// TIA Portal project "Tesis_Aeroponicos_V1" (V15.1)

(* hardware
DEVICE "S7300/ET200M station_1"  S7-300 station
   slot 0: "Rail_0"  Rail  6ES7 390-1***0-0AA0
   slot 2: "PLC_1"  CPU 313C  6ES7 313-5BF03-0AB0  V2.6
      slot 0: "MPI interface_1"  X1
      slot 2: "DI 24/DO 16_1"  DI24/DO16
      slot 3: "AI 5/AO 2_1"  AI5/AO2
      slot 4: "Count_1"  Counter
   slot 4: "CP 343-1 Advanced-IT_1"  CP 343-1 ADVANCED-IT  6GK7 343-1GX30-0XE0  V1.2
*)

// ===== PLC "PLC_1"  CPU 313C =====

VAR_GLOBAL   // PLC tag table "Default tag table"
   "E/S LoRa" AT %IW752 : Int;
   "E/S Valvula" AT %QW752 : Int;
   "D_valvula" AT %Q124.0 : Bool;
   "IO_1" AT %I124.0 : Bool;
   "Tag_1" AT %MW1 : Int;
   "Salida" AT %MD4 : Real;
   "Flag2" AT %M0.0 : Bool;
   "Entero" AT %MW8 : Int;
   "Tag_2" AT %M0.1 : Bool;
   "Test" AT %Q124.1 : Bool;
   "Control_temp" AT %Q125.7 : Bool;
   "Tag_3" AT %MD12 : Real;
   "Riego_45" AT %Q125.6 : Bool;
   "Riego_30" AT %Q125.5 : Bool;
   "Riego_15" AT %Q125.4 : Bool;
   "Tag_4" AT %T0 : Timer;
   "Tag_5" AT %T1 : Timer;
   "Tag_6" AT %M0.2 : Bool;
   "Tag_7" AT %M0.3 : Bool;
   "Tag_8" AT %M0.4 : Bool;
   "Tag_9" AT %M0.5 : Bool;
   "Tag_10" AT %T2 : Timer;
   "Tag_11" AT %T3 : Timer;
   "Tag_12" AT %MW6 : Word;
   "Tag_13" AT %M0.6 : Bool;
   "Tag_14" AT %M0.7 : Bool;
END_VAR

// folder: SystemBlocksFolder/ReportSystemErrorFolder

DATA_BLOCK "RSE_DIAGNOSTIC_STATUS_DB"   // DB127
TITLE = Bloque de diagnóstico Notificar errores del sistema
{ S7_Optimized_Access := 'FALSE' }
AUTHOR : SIMATIC
FAMILY : RSEDIAG
NAME : RSE7
VERSION : 1.0
// Este DB forma parte de Notificar errores de sistema y es actualizado por el FB de Notificar errores de sistema.
//  Es una interfaz para asistir el diagnóstico de sistema a través del CPU Webserver.
   VAR
      Directory : Struct
         D_Version : Word := WORD#16#0100;   // Versión que soporta 'Notificar errores de sistema' (SFM)
         D_pGlobalState : Word := WORD#16#0010;   // Offset de byte hasta el principio de la parte "GlobalState"
         D_pQuery : Word := WORD#16#0014;   // Offset de byte hasta el principio de la parte "Query"
         D_pComponent : Word := WORD#16#0020;   // Offset de byte hasta el principio de la parte "Component"
         D_pError : Word := WORD#16#0024;   // Offset de byte hasta el principio de la parte "Error"
         D_pState : Word := WORD#16#0028;   // Offset de byte hasta el principio de la parte "State"
         D_pAlarm : Word := WORD#16#005A;   // Offset de byte hasta el principio de la parte "Alarm"
         D_pSubComponent : Word := WORD#16#0082;   // Offset de byte hasta el principio de la parte "Subcomponent"
      END_STRUCT;
      GlobalState : Struct
         G_EventCount : Word := WORD#16#0000;   // ID del último evento (contador)
         G_StartReporting : Bool := FALSE;   // Evaluando el arranque
      END_STRUCT;
      Query : Struct
         Q_ClientID_User : DWord := DWORD#16#0000_0000;   // ID del cliente
         Q_ClientID_Intern : DWord := DWORD#16#0000_0000;   // ID del cliente (interno)
         Q_WithSubComponent : Bool := FALSE;   // Con/sin estado de los subcomponentes (más lento)
         Q_SubComponentAlarm : Bool := FALSE;   // AS-iMaster gibt AS-iSlave Alarme zurück
         Q_Reserved2 : Bool := FALSE;   // Reservado
         Q_Reserved3 : Bool := FALSE;   // Reservado
         Q_Reserved4 : Bool := FALSE;   // Reservado
         Q_Reserved5 : Bool := FALSE;   // Reservado
         Q_Reserved6 : Bool := FALSE;   // Reservado
         Q_Reserved7 : Bool := FALSE;   // Reservado
         Q_Start : Bool := FALSE;   // Iniciar consulta
         Q_Error : Byte := BYTE#16#00;   // Error interno en la consulta
         Q_Reserved8 : Byte := BYTE#16#00;   // Reservado
      END_STRUCT;
      Component : Struct
         C_AddressMode : Byte := BYTE#16#00;   // Modo de direccionamiento del módulo
         C_Reserved1 : Byte := BYTE#16#00;   // Reservado
         C_ComponentID : Word := WORD#16#0000;   // ID de hardware del componente (interno)
      END_STRUCT;
      Error : Struct
         E_ErrorNo : Word := WORD#16#0000;   // Índice del error solicitado/efectivo
         E_LastError : Bool := FALSE;   // TRUE, si E_ErrorNo contiene el índice del último error, de lo contrario FALSE
      END_STRUCT;
      State : Struct
         S_Hierarchy : Byte := BYTE#16#00;   // Reservado
         S_Periphery : Byte := BYTE#16#00;   // Reservado
         S_SupFault : Bool := FALSE;   // No se puede acceder al componente
         S_NotAvailable : Bool := FALSE;   // El componente no existe
         S_Faulty : Bool := FALSE;   // El componente falla; la parte "Alarm" no está vacía
         S_MoreErrors : Bool := FALSE;   // Hay más errores de los que puede guardar 'Notificar errores de sistema' (SFM).
         S_Maintenance1 : Bool := FALSE;   // Mantenimiento necesario pendiente
         S_Maintenance2 : Bool := FALSE;   // Mantenimiento solicitado pendiente
         S_Deactivated : Bool := FALSE;   // The component was deactivated
         S_Reserved2 : Bool := FALSE;   // Reservado
         S_SubFault : Bool := FALSE;   // Fallo en un subcomponente
         S_SubMaintenance1 : Bool := FALSE;   // Mantenimiento necesario de un subcomponente
         S_SubMaintenance2 : Bool := FALSE;   // Mantenimiento solicitado para un subcomponente
         S_SubDeactivated : Bool := FALSE;   // At least one lower-level component is disabled
         S_Reserved4 : Bool := FALSE;   // Reservado
         S_Reserved5 : Bool := FALSE;   // Reservado
         S_Reserved6 : Bool := FALSE;   // Reservado
         S_Reserved7 : Bool := FALSE;   // Reservado
         S_TIAMS : DWord := DWORD#16#0000_0000;   // Estado de mantenimiento del componente
         S_TIAMSChannelExist : DWord := DWORD#16#0000_0000;   // Estado de mantenimiento: canales configurados
         S_TIAMSChannelOK : DWord := DWORD#16#0000_0000;   // Estado de mantenimiento: canales que fallan
         S_ChannelCount : Word := WORD#16#0000;   // Número de canales; solo es válido si está activado Q_WithSubComponent
         S_ChannelVector : Array[0..255] of Bool;   // Lista de canales afectados; sólo es válida si está activado Q_WithSubComponent
      END_STRUCT;
      Alarm : Struct
         A_ComponentID : Word := WORD#16#0000;   // ID de hardware del componente (interna)
         A_TextID1 : Word := WORD#16#0000;   // ID del primer texto de error
         A_TextLexikonID1 : Word := WORD#16#0000;   // ID de la primera librería de textos de error
         A_HelpTextLexikonID1 : Word := WORD#16#0000;   // ID de la primera librería de textos de ayuda
         A_MapTextID : Word := WORD#16#0000;   // ID del primer texto de error en el archivo de exportación (HMI)
         A_MapHelpTextID : Word := WORD#16#0000;   // ID del primer texto de ayuda en el archivo de exportación (HMI)
         A_TextID2 : Word := WORD#16#0000;   // ID del segundo texto de error
         A_TextLexikonID2 : Word := WORD#16#0000;   // ID de la segunda librería de textos de error
         A_HelpTextLexikonID2 : Word := WORD#16#0000;   // ID de la segunda librería de textos de ayuda
         A_MapTextID2 : Word := WORD#16#0000;   // ID del segundo texto de error en el archivo de exportación (HMI)
         A_MapHelpTextID2 : Word := WORD#16#0000;   // ID del segundo texto de ayuda en el archivo de exportación (HMI)
         A_AlarmID : DWord := DWORD#16#0000_0000;   // Número de aviso
         A_ValueCount : Word := WORD#16#000C;   // Cantidad de los demás bytes ocupados
         A_AssociatedValue : Array[1..6] of Word;   // Valores asociados del aviso
      END_STRUCT;
      SubComponent : Struct
         U_SubComponentCount : Word := WORD#16#0000;   // Número de subcomponentes
         U_SubComponentFault : Array[1..8] of Byte;   // Lista del estado de los componentes subordinados, 1 byte por componente
      END_STRUCT;
   END_VAR
BEGIN
END_DATA_BLOCK

// folder: (top level)

ORGANIZATION_BLOCK "Main"   // OB1, LAD
TITLE = "Main Program Sweep (Cycle)"
{ S7_Optimized_Access := 'FALSE' }
VERSION : 0.1
   VAR_TEMP
      OB1_EV_CLASS : Byte;   // Bits 0-3 = 1 (Coming event), Bits 4-7 = 1 (Event class 1)
      OB1_SCAN_1 : Byte;   // 1 (Cold restart scan 1 of OB 1), 3 (Scan 2-n of OB 1)
      OB1_PRIORITY : Byte;   // Priority of OB Execution
      OB1_OB_NUMBR : Byte;   // 1 (Organization block 1, OB1)
      OB1_RESERVED_1 : Byte;   // Reserved for system
      OB1_RESERVED_2 : Byte;   // Reserved for system
      OB1_PREV_CYCLE : Int;   // Cycle time of previous OB1 scan (milliseconds)
      OB1_MIN_CYCLE : Int;   // Minimum cycle time of OB1 (milliseconds)
      OB1_MAX_CYCLE : Int;   // Maximum cycle time of OB1 (milliseconds)
      OB1_DATE_TIME : Date_And_Time;   // Date and time OB1 started
      flag : Bool;
      Fallo : Word;
   END_VAR
BEGIN

REGION Network 1
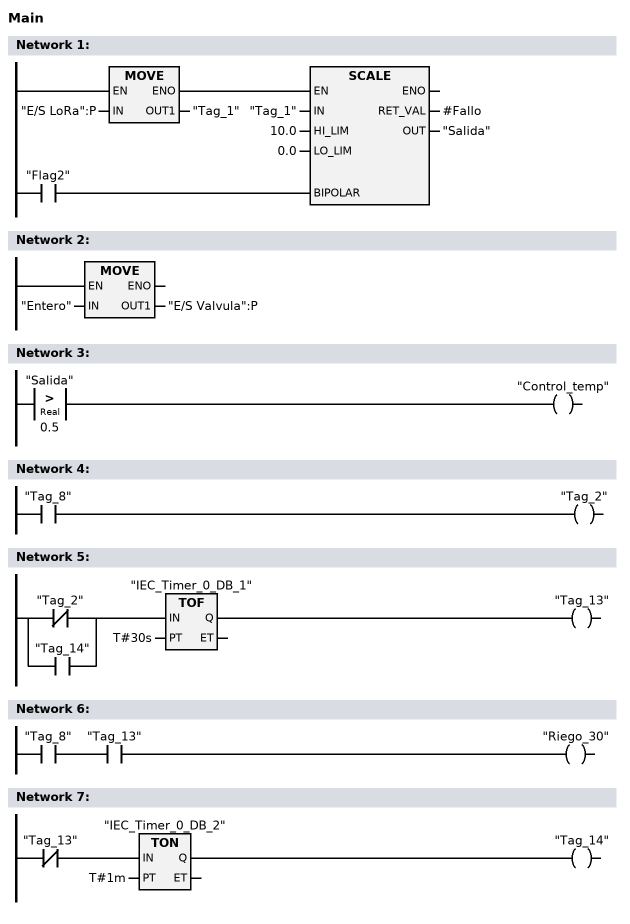
   // ENO of a box is taken as its EN; it also drops when the box reports an error
   "Tag_1" := "E/S LoRa":P;
   #Fallo := SCALE(IN := "Tag_1", HI_LIM := 10.0, LO_LIM := 0.0, BIPOLAR := "Flag2", OUT => "Salida");
END_REGION

REGION Network 2
   RUNG wire#powerrail
      { S7_GenerateENO := "TRUE" } Move(in := "Entero", out1 => "E/S Valvula":P)
   END_RUNG
   // the same network as SCL:
   "E/S Valvula":P := "Entero";
END_REGION

REGION Network 3
   RUNG wire#powerrail
      { S7_Templates := "SrcType := Real" } GT_Contact(in1 := "Salida", in2 := 0.5)
      Coil( "Control_temp" )
   END_RUNG
   // the same network as SCL:
   "Control_temp" := "Salida" > 0.5;
END_REGION

REGION Network 4
   RUNG wire#powerrail
      Contact( "Tag_8" )
      Coil( "Tag_2" )
   END_RUNG
   // the same network as SCL:
   "Tag_2" := "Tag_8";
END_REGION

REGION Network 5
   "IEC_Timer_0_DB_1".TOF(IN := NOT "Tag_2" OR "Tag_14", PT := T#30s);
   "Tag_13" := "IEC_Timer_0_DB_1".Q;
END_REGION

REGION Network 6
   RUNG wire#powerrail
      Contact( "Tag_8" )
      Contact( "Tag_13" )
      Coil( "Riego_30" )
   END_RUNG
   // the same network as SCL:
   "Riego_30" := "Tag_8" AND "Tag_13";
END_REGION

REGION Network 7
   "IEC_Timer_0_DB_2".TON(IN := NOT "Tag_13", PT := T#1m);
   "Tag_14" := "IEC_Timer_0_DB_2".Q;
END_REGION
END_ORGANIZATION_BLOCK

ORGANIZATION_BLOCK "I/O_FLT1"   // OB82, STL
TITLE = "I/O Point Fault"
{ S7_Optimized_Access := 'FALSE' }
VERSION : 0.1
   VAR_TEMP
      OB82_EV_CLASS : Byte;   // 16#39, Event class 3, Entering event state, Internal fault event
      OB82_FLT_ID : Byte;   // 16#XX, Fault identifcation code
      OB82_PRIORITY : Byte;   // Priority of OB Execution
      OB82_OB_NUMBR : Byte;   // 82 (Organization block 82, OB82)
      OB82_RESERVED_1 : Byte;   // Reserved for system
      OB82_IO_FLAG : Byte;   // Input (01010100), Output (01010101)
      OB82_MDL_ADDR : Word;   // Base address of module with fault
      OB82_MDL_DEFECT : Bool;   // Module defective
      OB82_INT_FAULT : Bool;   // Internal fault
      OB82_EXT_FAULT : Bool;   // External fault
      OB82_PNT_INFO : Bool;   // Point information
      OB82_EXT_VOLTAGE : Bool;   // External voltage low
      OB82_FLD_CONNCTR : Bool;   // Field wiring connector missing
      OB82_NO_CONFIG : Bool;   // Module has no configuration data
      OB82_CONFIG_ERR : Bool;   // Module has configuration error
      OB82_MDL_TYPE : Byte;   // Type of module
      OB82_SUB_MDL_ERR : Bool;   // Sub-Module is missing or has error
      OB82_COMM_FAULT : Bool;   // Communication fault
      OB82_MDL_STOP : Bool;   // Module is stopped
      OB82_WTCH_DOG_FLT : Bool;   // Watch dog timer stopped module
      OB82_INT_PS_FLT : Bool;   // Internal power supply fault
      OB82_PRIM_BATT_FLT : Bool;   // Primary battery is in fault
      OB82_BCKUP_BATT_FLT : Bool;   // Backup battery is in fault
      OB82_RESERVED_2 : Bool;   // Reserved for system
      OB82_RACK_FLT : Bool;   // Rack fault, only for bus interface module
      OB82_PROC_FLT : Bool;   // Processor fault
      OB82_EPROM_FLT : Bool;   // EPROM fault
      OB82_RAM_FLT : Bool;   // RAM fault
      OB82_ADU_FLT : Bool;   // ADU fault
      OB82_FUSE_FLT : Bool;   // Fuse fault
      OB82_HW_INTR_FLT : Bool;   // Hardware interupt input in fault
      OB82_RESERVED_3 : Bool;   // Reserved for system
      OB82_DATE_TIME : Date_And_Time;   // Date and time OB82 started
   END_VAR
BEGIN

REGION Network 1: Llamar bloque de diagnóstico de sistema
         CALL  "RSE_FB", "RSE_DB";
END_REGION
END_ORGANIZATION_BLOCK

ORGANIZATION_BLOCK "OBNL_FLT"   // OB85, STL
TITLE = "Organization Block (OB) Not Loaded Fault"
{ S7_Optimized_Access := 'FALSE' }
VERSION : 0.1
   VAR_TEMP
      OB85_EV_CLASS : Byte;   // 16#35 Event class 3
      OB85_FLT_ID : Byte;   // 16#XX, Fault identification code
      OB85_PRIORITY : Byte;   // Priority of OB Execution
      OB85_OB_NUMBR : Byte;   // 85 (Organization block 85, OB85)
      OB85_RESERVED_1 : Byte;   // Reserved for system
      OB85_RESERVED_2 : Byte;   // Reserved for system
      OB85_RESERVED_3 : Int;   // Reserved for system
      OB85_ERR_EV_CLASS : Byte;   // Class of event causing error
      OB85_ERR_EV_NUM : Byte;   // Number of event causing error
      OB85_OB_PRIOR : Byte;   // Priority of OB causing error
      OB85_OB_NUM : Byte;   // Number of OB causing error
      OB85_DATE_TIME : Date_And_Time;   // Date and time OB85 started
   END_VAR
BEGIN

REGION Network 1
         L     b#16#A1;  //
         L     #OB85_FLT_ID;
         ==I;
         JC    K_OB;
         L     b#16#A2;  //
         ==I;
         JC    K_OB;
         L     b#16#A3;  //
         L     #OB85_FLT_ID;
         ==I;
         JC    K_B;
         JU    F_PA;
END_REGION

REGION Network 2
   K_OB: JU    STOP;
         JU    ENDE;
END_REGION

REGION Network 3
   K_B:  JU    STOP;
         JU    ENDE;
END_REGION

REGION Network 4
   F_PA: NOP   0;
         JU    ENDE;
END_REGION

REGION Network 5
   STOP: CALL  STP;
END_REGION

REGION Network 6

   //

   ENDE: NOP   0;
END_REGION
END_ORGANIZATION_BLOCK